// TwinCAT 3 PLC project motion_supplement_test
// ProgramVersion: 3.1.4026.16
// libraries:
//   [Nepionic Motion Supplement], * (Nepionic)
//   Tc2_MC2, * (Beckhoff Automation GmbH)
//   Tc2_Standard, * (Beckhoff Automation GmbH)
//   Tc2_System, * (Beckhoff Automation GmbH)
// project tree:
//   Programs/ Test.TcPOU
//   Tasks/ PlcTask.TcTTO
// real-time tasks:
//   TASK PlcTask: cycle T#10ms, priority 20, ADS port 350
// motion (NC):
//   TASK NC-Task 1 SAF: cycle T#2ms, priority 4, ADS port 501
//   TASK NC-Task 1 SVB: cycle T#10ms, priority 8, ADS port 511
//   AXIS Axis 1 (id 1)
//     OtherSettings: AllowMotionCmdToSlave=true
//     encoder EncType=1
//     drive DrvType=5
//       Analog: TorqueSetpointScale=10, ScaleFactorActTorque=0.1
//       TimeComp: TaskDelayCycles=1
//     controller CtrType=1
//       CtrPara: PriorControlFactor=1
//         Observer: BandWidth=20
// variable links:
//   motion_supplement_test/motion_supplement_test Instance <-> NC-Task 1 SAF/Axes/Axis 1
//     PlcTask Inputs/Main.axis_ref.NcToPlc <-> Outputs/ToPlc
//     PlcTask Outputs/Main.axis_ref.PlcToNc <-> Inputs/FromPlc

CONFIGURATION motion_supplement_test
    RESOURCE PLC ON TwinCAT3
        TASK PlcTask(INTERVAL := T#10ms, PRIORITY := 20);
        PROGRAM Test WITH PlcTask : Test;
    END_RESOURCE
END_CONFIGURATION

// ---- Programs/Test.TcPOU
PROGRAM Test
VAR
	axis_ref : Axis_Ref;
	power : Mc_Power;
	reset : Mc_Reset;
	stop : Mc_Stop;
	move_velocity : Mc_MoveVelocity;
	move_continuous_velocity : Mc_MoveContinuousVelocity;
	enable : BOOL;
	perform_reset : BOOL;
	perform_stop : BOOL;
	
	perform_move_velocity : BOOL;
	perform_move_continuous_velocity : BOOL;
	move_velocity_speed : LREAL := 5.0;
END_VAR

power(
	Axis := axis_ref,
	Enable := enable,
	Enable_Positive := enable,
	Enable_Negative := enable,
	Override := 100.0,
	BufferMode := Mc_BufferMode.Mc_Aborting
);

reset(
	Axis := axis_ref,
	Execute := perform_reset
);

IF NOT reset.Busy AND NOT reset.Error THEN
	perform_reset := FALSE;
END_IF

stop(
	Axis := axis_ref,
	Execute := perform_stop
);

IF NOT stop.Done THEN
	perform_stop := FALSE;
END_IF

move_velocity(
	Axis := axis_ref,
	Execute := perform_move_velocity,
	Velocity := move_velocity_speed,
	Direction := Mc_Direction.Mc_Positive_Direction
);

IF NOT move_velocity.Busy AND NOT move_velocity.Error THEN
	perform_move_velocity := FALSE;
END_IF

move_continuous_velocity(
	Axis := axis_ref,
	Execute := perform_move_continuous_velocity,
	Velocity := move_velocity_speed,
	Direction := Mc_Direction.Mc_Positive_Direction
);

END_PROGRAM
